FUNCTION_BLOCK Test_AssertEquals_UINT EXTENDS T_UnitTestBase
VAR
    AssertionUnderTest : T_Assertion;
    UINT_Variable : UINT := 1111;
END_VAR

// Test the assertion...
AssertionUnderTest.AssertEquals_UINT(
    Expected := 2222,
    Actual   := UINT_Variable,
    VariableName := 'UINT_Variable');
   
// Assert that the assertion failed...
Assertion.AssertEquals_BOOL(Expected     := TRUE,
                            Actual       := AssertionUnderTest.AssertionFailed,
                            VariableName := 'AssertionUnderTest.AssertionFailed');

// Check the assertion worked...  
CheckAssertion(NextState := 0);

END_FUNCTION_BLOCK

(* stored: Version 1.1.0.1, ProductVersion 3.1.4024.11
   POU Test_AssertEquals_UINT: Id {7be0dfef-0c15-47b8-a422-f4c2311ff565}, SpecialFunc None *)
